// TIA Portal V20 export
FUNCTION_BLOCK "Simulation_addon"   // FB23, LAD
// stored: Access Published, MemoryReserve 100, SetENOAutomatically false
   VAR_INPUT
      cmdHomePos : Bool;
      cmdWorkPos : Bool;
   END_VAR
   VAR_OUTPUT
      homePos : Bool;
      WorkPos : Bool;
   END_VAR
   VAR
      IEC_Timer_0_Instance { S7_SetPoint := 'True'} : TON_TIME;
      IEC_Timer_0_Instance_1 { S7_SetPoint := 'True'} : TON_TIME;
   END_VAR
   VAR CONSTANT
      delayTime : Time := T#100ms;
   END_VAR
BEGIN

REGION Network 1
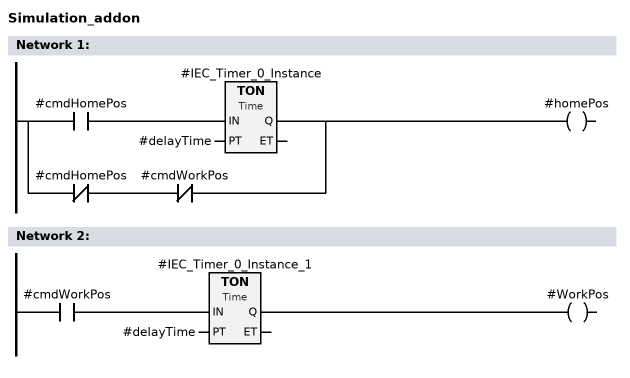
   RUNG wire#powerrail
      Contact( #cmdHomePos )
      { S7_Templates := "time_type := Time" } #IEC_Timer_0_Instance.TON(pt := #delayTime, et =>)
      wire#w1
      Coil( #homePos )
   END_RUNG
   RUNG wire#powerrail
      I_Contact( #cmdHomePos )
      I_Contact( #cmdWorkPos )
   END_RUNG wire#w1
   // the same network as SCL:
   #IEC_Timer_0_Instance(IN := #cmdHomePos, PT := #delayTime);   // TON
   #homePos := #IEC_Timer_0_Instance.Q OR (NOT #cmdHomePos AND NOT #cmdWorkPos);
END_REGION

REGION Network 2
   RUNG wire#powerrail
      Contact( #cmdWorkPos )
      { S7_Templates := "time_type := Time" } #IEC_Timer_0_Instance_1.TON(pt := #delayTime, et =>)
      Coil( #WorkPos )
   END_RUNG
   // the same network as SCL:
   #IEC_Timer_0_Instance_1(IN := #cmdWorkPos, PT := #delayTime);   // TON
   #WorkPos := #IEC_Timer_0_Instance_1.Q;
END_REGION
END_FUNCTION_BLOCK
